{attribute 'GeneratedUsingTerminal: EL3204-0000-0016'}
{attribute addProperty BoxType "EL3204-0000-0016"}
{attribute addProperty Id "EtcSlaveTerminalBaseRTD_Inputs_Channel_1AT %I*RTD_Inputs_Channel_EA9DF21E9RTD_Inputs_Channel_2AT %I*RTD_Inputs_Channel_EA9DF21E9RTD_Inputs_Channel_3AT %I*RTD_Inputs_Channel_EA9DF21E9RTD_Inputs_Channel_4AT %I*RTD_Inputs_Channel_EA9DF21E9WcStateAT %I*WcState_9091E0EB2InfoDataAT %I*InfoData_32EB74EA10"}
{attribute addProperty CRC "1263763227"}
{attribute addProperty Size "48"}
TYPE EL3204_4B537F1B EXTENDS EtcSlaveTerminalBase :
STRUCT
	{attribute addProperty Name "RTD_Inputs_Channel_1"}
	RTD_Inputs_Channel_1 : RTD_Inputs_Channel_EA9DF21E;
	{attribute addProperty Name "RTD_Inputs_Channel_2"}
	RTD_Inputs_Channel_2 : RTD_Inputs_Channel_EA9DF21E;
	{attribute addProperty Name "RTD_Inputs_Channel_3"}
	RTD_Inputs_Channel_3 : RTD_Inputs_Channel_EA9DF21E;
	{attribute addProperty Name "RTD_Inputs_Channel_4"}
	RTD_Inputs_Channel_4 : RTD_Inputs_Channel_EA9DF21E;
	{attribute addProperty Name "WcState"}
	WcState : WcState_9091E0EB;
	{attribute addProperty Name "InfoData"}
	InfoData : InfoData_32EB74EA;
END_STRUCT
END_TYPE

(* stored: Version 1.2.0.0, ProductVersion 3.1.4024.9
   DUT EL3204_4B537F1B: Id {822b693e-c050-4f9a-b039-b00bc5ac4624} *)
